// TwinCAT 3 PLC project Pneumatiek_test
// ProgramVersion: 3.1.4024.0
// libraries:
//   Tc2_MC2, * (Beckhoff Automation GmbH)
//   Tc2_Standard, * (Beckhoff Automation GmbH)
//   Tc2_System, * (Beckhoff Automation GmbH)
//   Tc3_Module, * (Beckhoff Automation GmbH)
// project tree:
//   / PlcTask.TcTTO
//   POUs/ MAIN.TcPOU

CONFIGURATION Pneumatiek_test
    RESOURCE PLC ON TwinCAT3
        TASK PlcTask(INTERVAL := T#10ms, PRIORITY := 23);
        PROGRAM MAIN WITH PlcTask : MAIN;
    END_RESOURCE
END_CONFIGURATION

// ---- POUs/MAIN.TcPOU
PROGRAM MAIN
VAR
	knop_start AT %I*: BOOL;
	knop_stop AT %I*: BOOL;
	knop_reset AT %I*: BOOL;
	druk_uit AT %Q*: BOOL;
	druk_in AT %Q*: BOOL;
	z_in AT %Q*: BOOL;
	z_uit AT %Q*: BOOL;
	gripper_in AT %Q*: BOOL;
	gripper_uit AT %Q*: BOOL;
	vacuum AT %Q*: BOOL;
	state: INT := 0;
	Yas: AXIS_REF;
	YMotorPower: MC_power;
	YMotorPosition: MC_MoveAbsolute;
	YMotorHome: MC_Home;
	YMotorJog: MC_Jog;
	picktimer: TON;
	lamp_rood AT %Q*: BOOL;
	lamp_oranje AT %Q*: BOOL;
	lamp_groen AT %Q*: BOOL;
	lamp_blauw AT %Q*: BOOL;
END_VAR


YMotorPosition(Axis := Yas, Velocity := 1300, Acceleration := 5000, Deceleration := 5000, Jerk := 100000);
YMotorPower(Axis := Yas, Enable := TRUE, Enable_Positive := TRUE, Enable_Negative := TRUE);
CASE state OF

0 : z_in := TRUE;
	gripper_uit := TRUE;
	gripper_in := FALSE;
	lamp_groen := TRUE;
	IF knop_reset = TRUE THEN
		YMotorHome(Axis := Yas, Execute := TRUE, Position := 0, HomingMode := MC_DIRECT);
	END_IF
	IF YMotorHome.Done = TRUE THEN
		state := 1;
	END_IF






1 :	YMotorHome(Axis := Yas, Execute := FALSE);
	IF knop_start = TRUE THEN
		YMotorPosition(Axis := Yas, Execute := TRUE, Position := 295);
	END_IF	
	IF YMotorPosition.Done = TRUE THEN
		z_in := FALSE;
		gripper_in := TRUE;
		z_uit := TRUE;
		vacuum := TRUE;
		picktimer(IN := TRUE, PT := T#3S);
	END_IF
	IF picktimer.Q = TRUE THEN
		
		z_uit := FALSE;
		gripper_in := FALSE;
		z_in := TRUE;
		gripper_uit := TRUE;
		state := 2;
	END_IF
2 : YMotorPosition(Axis := Yas, Execute := FALSE); 
	state := 3;
	
3 :	YMotorPosition(Axis := Yas, Execute := TRUE, Position := 6562); 
		picktimer(IN := FALSE);
		IF YMotorPosition.Done = TRUE THEN
		    YMotorPosition(Axis := Yas, Execute := FALSE);
			z_in := FALSE;
			z_uit := TRUE;
		END_IF
		
		IF z_uit = TRUE THEN
			vacuum := FALSE;
		END_IF
		
		IF vacuum = FALSE THEN
			z_uit := FALSE;
			z_in := TRUE;
			state := 1;
		END_IF
	
		
	
END_CASE

END_PROGRAM
